TYPE LogicalInterlockSubstate :
STRUCT
	recipeEnableSubstate : ARRAY[1..GVL_CONSTANT.NumInterlockRecipeEnableSubstate] OF BOOL;
	openReactorSubstate : ARRAY[1..GVL_CONSTANT.NumInterlockOpenReactorSubstate] OF BOOL;
END_STRUCT
END_TYPE

(* stored: Version 1.1.0.1, ProductVersion 3.1.4026.11
   DUT LogicalInterlockSubstate: Id {1cf4387c-9c9c-4486-8b62-3269d0748222} *)
